// TIA Portal V17 export
// export: Created 2023-04-03T06:31:43.3625414Z, ExportSetting WithDefaults, DisplayName Totally Integrated Automation Portal, DisplayVersion V17 Update 4, DisplayName TIA Portal Openness, DisplayVersion V17 Update 4, DisplayName TIA Portal Version Control Interface, DisplayVersion V17, DisplayName STEP 7 Professional, DisplayVersion V17 Update 4, DisplayName STEP 7 Safety, DisplayVersion V17, DisplayName WinCC Professional, DisplayVersion V17 Update 4
TYPE "R_PE_1"
// stored: IsFailsafeCompliant false
   STRUCT
      rPacMeas : Real := 0.0;   // Array1 [1] - SV1.7 / 41001
      rQacMeas : Real := 0.0;   // Array1 [2] - SV1.8 / 41002
      rSacMeas : Real := 0.0;   // Array1 [3] - SV1.9 / 41003
      rPFmeas : Real := 0.0;   // Array1 [4] - SV1.10 / 41004
      rFrMeas : Real := 0.0;   // Array1 [5] - SV1.11 / 41005
      rVrsMeas : Real := 0.0;   // Array1 [6] - SV1.1 / 41006
      rVstMeas : Real := 0.0;   // Array1 [7] - SV1.2 / 41007
      rVtrMeas : Real := 0.0;   // Array1 [8] - SV1.3 / 41008
      rIrMeas : Real := 0.0;   // Array1 [9] - SV1.4 / 41009
      rIsMeas : Real := 0.0;   // Array1 [10] - SV1.5 / 41010
      rItMeas : Real := 0.0;   // Array1 [11] - SV1.6 / 41011
      rPdcMeas : Real := 0.0;   // Array1 [12] - SV2.5 / 41013
      rIdcMeas : Real := 0.0;   // Array1 [13] - SV2.6 / 41014
      iImonDc1St : Int := 0;   // Array1 [14] - SV3.2.1 / 41015
      iImonAcSt : Int := 0;   // Array1 [15] - SV3.1.1 / 41021
      iCodeFlt : Int := 0;   // Array1 [16] - SV4.1.1 / 41026
      iCodeWarn : Int := 0;   // Array1 [17] - SV4.1.2 / 41027
      iCodeSt : Int := 0;   // Array1 [18] - SV4.1.3 / 41028
      xInvOffSt : Bool;
      xInvStandBySt : Bool;
      xInvReadySt : Bool;
      xInvPrOnSt : Bool;
      xInvRunSt : Bool;
      xInvStopSt : Bool;
      xInvFltSt : Bool;
      rTmodAcMeas : Real := 0.0;   // Array1 [19] - SV4.1.4 / 41029
      rTigbtMaxMeas : Real := 0.0;   // Array1 [20] - SV4.1.5 / 41030
      rTmodMaxMeas : Real := 0.0;   // Array1 [21] - SV4.1.6 / 41031
      wDIboardSt : Word := 0;   // 41032 / Array1 [22] - SV4.1.7
      wDOboardSt : Word := 0;   // 41033 / Array1 [23] - SV4.1.8
      rTmodAcInMeas : Real := 0.0;   // 41034 / Array1 [24] - SV4.1.9
      iFltModId : Int := 0;   // 41036 / Array1 [25] - SV4.1.1b
      rRHintMeas : Real := 0.0;   // 41037 / Array1 [26] - SV4.1.11
      rVaux1Meas : Real := 0.0;   // 41039 / Array1 [27] - SV4.1.14
      rVaux2Meas : Real := 0.0;   // 41040 / Array1 [28] - SV4.1.15
      rPacAvlLim : Real := 0.0;   // Array1 [29] - SV4.2.1 / 41141
      rQacAvlLim : Real := 0.0;   // Array1 [30] - SV4.2.2 / 41142
      wDUchanSel : Word := 0;   // Array1 [31] - SV10.1 / 41251
      rVdcBus1Meas : Real := 0.0;   // Array1 [32] - SV2.1.1 / 47402
      rVdcBus2Meas : Real := 0.0;   // Array1 [33] - SV2.1.2 / 47402
      rIdcBus1Meas : Real := 0.0;   // Array1 [34] - SV2.6a / 47410
      rIdcBus2Meas : Real := 0.0;   // Array1 [35] - SV2.6b / 47411
      rIRFIcapRef : Real := 0.0;   // Array1 [36] - SV2.11 / 47416
      rPavlChaBus1 : Real;   // Array1 [37] - SV4.2.1a
      rPavlDschBus1 : Real;   // Array1 [38] - SV4.2.1b
      rPavlChaBus2 : Real;   // Array1 [39] - SV4.2.1c
      rPavlDschBus2 : Real;   // Array1 [40] - SV4.2.1d
      iImonDc2St : Int := 0;   // Array1 [41] - SV3.3.1 / 41015
      wDUchanSt : Word;   // Array1 [42] - SV10.10
      wMod1St : Int;   // Array1 [43]
      xMod1StopSt : Bool;
      xMod1ReadySt : Bool;
      xMod1MainAcSt : Bool;
      xMod1RunSt : Bool;
      xMod1FltSt : Bool;
      rMod1PacMeas : Real;   // Array1 [44]
      rMod1QacMeas : Real;   // Array1 [45]
      wMod1IOSt : Word;   // Array1 [46]
      xMod1ThermLCLst : Bool;
      xMod1FanSt : Bool;
      xMod1AcMainSt : Bool;
      xMod1AcSoftChaSt : Bool;
      xMod1LCLst : Bool;
      xMod1DcSwitchSt : Bool;
      rMod1TempR1Meas : Real;   // Array1 [47]
      rMod1TempR2Meas : Real;   // Array1 [48]
      rMod1TempR3Meas : Real;   // Array1 [49]
      rMod1TempS1Meas : Real;   // Array1 [50]
      rMod1TempS2Meas : Real;   // Array1 [51]
      rMod1TempS3Meas : Real;   // Array1 [52]
      rMod1TempT1Meas : Real;   // Array1 [53]
      rMod1TempT2Meas : Real;   // Array1 [54]
      rMod1TempT3Meas : Real;   // Array1 [55]
      wMod2St : Int;   // Array1 [56]
      xMod2StopSt : Bool;
      xMod2ReadySt : Bool;
      xMod2MainAcSt : Bool;
      xMod2RunSt : Bool;
      xMod2FltSt : Bool;
      rMod2PacMeas : Real;   // Array1 [57]
      rMod2QacMeas : Real;   // Array1 [58]
      wMod2IOSt : Word;   // Array1 [59]
      xMod2ThermLCLst : Bool;
      xMod2FanSt : Bool;
      xMod2AcMainSt : Bool;
      xMod2AcSoftChaSt : Bool;
      xMod2LCLst : Bool;
      xMod2DcSwitchSt : Bool;
      rMod2TempR1Meas : Real;   // Array1 [60]
      rMod2TempR2Meas : Real;   // Array1 [61]
      rMod2TempR3Meas : Real;   // Array1 [62]
      rMod2TempS1Meas : Real;   // Array1 [63]
      rMod2TempS2Meas : Real;   // Array1 [64]
      rMod2TempS3Meas : Real;   // Array1 [65]
      rMod2TempT1Meas : Real;   // Array1 [66]
      rMod2TempT2Meas : Real;   // Array1 [67]
      rMod2TempT3Meas : Real;   // Array1 [68]
      wMod3St : Int;   // Array1 [69]
      xMod3StopSt : Bool;
      xMod3ReadySt : Bool;
      xMod3MainAcSt : Bool;
      xMod3RunSt : Bool;
      xMod3FltSt : Bool;
      rMod3PacMeas : Real;   // Array1 [70]
      rMod3QacMeas : Real;   // Array1 [71]
      wMod3IOSt : Word;   // Array1 [72]
      xMod3ThermLCLst : Bool;
      xMod3FanSt : Bool;
      xMod3AcMainSt : Bool;
      xMod3AcSoftChaSt : Bool;
      xMod3LCLst : Bool;
      xMod3DcSwitchSt : Bool;
      rMod3TempR1Meas : Real;   // Array1 [73]
      rMod3TempR2Meas : Real;   // Array1 [74]
      rMod3TempR3Meas : Real;   // Array1 [75]
      rMod3TempS1Meas : Real;   // Array1 [76]
      rMod3TempS2Meas : Real;   // Array1 [77]
      rMod3TempS3Meas : Real;   // Array1 [78]
      rMod3TempT1Meas : Real;   // Array1 [79]
      rMod3TempT2Meas : Real;   // Array1 [80]
      rMod3TempT3Meas : Real;   // Array1 [81]
      wMod4St : Int;   // Array1 [82]
      xMod4StopSt : Bool;
      xMod4ReadySt : Bool;
      xMod4MainAcSt : Bool;
      xMod4RunSt : Bool;
      xMod4FltSt : Bool;
      rMod4PacMeas : Real;   // Array1 [83]
      rMod4QacMeas : Real;   // Array1 [84]
      wMod4IOSt : Word;   // Array1 [85]
      xMod4ThermLCLst : Bool;
      xMod4FanSt : Bool;
      xMod4AcMainSt : Bool;
      xMod4AcSoftChaSt : Bool;
      xMod4LCLst : Bool;
      xMod4DcSwitchSt : Bool;
      rMod4TempR1Meas : Real;   // Array1 [86]
      rMod4TempR2Meas : Real;   // Array1 [87]
      rMod4TempR3Meas : Real;   // Array1 [88]
      rMod4TempS1Meas : Real;   // Array1 [89]
      rMod4TempS2Meas : Real;   // Array1 [90]
      rMod4TempS3Meas : Real;   // Array1 [91]
      rMod4TempT1Meas : Real;   // Array1 [92]
      rMod4TempT2Meas : Real;   // Array1 [93]
      rMod4TempT3Meas : Real;   // Array1 [94]
      wMod5St : Int;   // Array1 [95]
      xMod5StopSt : Bool;
      xMod5ReadySt : Bool;
      xMod5MainAcSt : Bool;
      xMod5RunSt : Bool;
      xMod5FltSt : Bool;
      rMod5PacMeas : Real;   // Array1 [96]
      rMod5QacMeas : Real;   // Array1 [97]
      wMod5IOSt : Word;   // Array1 [98]
      xMod5ThermLCLst : Bool;
      xMod5FanSt : Bool;
      xMod5AcMainSt : Bool;
      xMod5AcSoftChaSt : Bool;
      xMod5LCLst : Bool;
      xMod5DcSwitchSt : Bool;
      rMod5TempR1Meas : Real;   // Array1 [99]
      rMod5TempR2Meas : Real;   // Array1 [100]
      rMod5TempR3Meas : Real;   // Array1 [101]
      rMod5TempS1Meas : Real;   // Array1 [102]
      rMod5TempS2Meas : Real;   // Array1 [103]
      rMod5TempS3Meas : Real;   // Array1 [104]
      rMod5TempT1Meas : Real;   // Array1 [105]
      rMod5TempT2Meas : Real;   // Array1 [106]
      rMod5TempT3Meas : Real;   // Array1 [107]
      wMod6St : Int;   // Array1 [108]
      xMod6StopSt : Bool;
      xMod6ReadySt : Bool;
      xMod6MainAcSt : Bool;
      xMod6RunSt : Bool;
      xMod6FltSt : Bool;
      rMod6PacMeas : Real;   // Array1 [109]
      rMod6QacMeas : Real;   // Array1 [110]
      wMod6IOSt : Word;   // Array1 [111]
      xMod6ThermLCLst : Bool;
      xMod6FanSt : Bool;
      xMod6AcMainSt : Bool;
      xMod6AcSoftChaSt : Bool;
      xMod6LCLst : Bool;
      xMod6DcSwitchSt : Bool;
      rMod6TempR1Meas : Real;   // Array1 [112]
      rMod6TempR2Meas : Real;   // Array1 [113]
      rMod6TempR3Meas : Real;   // Array1 [114]
      rMod6TempS1Meas : Real;   // Array1 [115]
      rMod6TempS2Meas : Real;   // Array1 [116]
      rMod6TempS3Meas : Real;   // Array1 [117]
      rMod6TempT1Meas : Real;   // Array1 [118]
      rMod6TempT2Meas : Real;   // Array1 [119]
      rMod6TempT3Meas : Real;   // Array1 [120]
   END_STRUCT;
END_TYPE
